FUNCTION_BLOCK Santino_Object EXTENDS TcoCore.TcoObject
VAR
	_francesca	:	AKid_Object(THIS^, TcoCore.NO.Structure);
	_kathryn 	:	AKid_Object(THIS^, TcoCore.NO.Structure);
	_frank		:	AKid_Object(THIS^, TcoCore.NO.Structure);
	_santino	:	AKid_Object(THIS^, TcoCore.NO.Structure);
END_VAR

END_FUNCTION_BLOCK

(* stored: Version 1.1.0.1, ProductVersion 3.1.4024.9
   POU Santino_Object: Id {1fcf27a4-725c-0efd-2dcd-a32ba27c10e9}, SpecialFunc None *)
